(* Logix 5000 project; controller Thurs_Lab2 vendor 1 type 14 code 156 rev 30.11; software revision 30.00 *)

TASK MainTask (continuous, watchdog 500 ms) : MainProgram

MODULES
   Local : vendor 1 type 14 code 156 (Compact 0, rev 30.11)
      DC_input : 1769-IQ16 (Compact 1, rev 1.1, Input RPI 20 ms)   // Dc input
           Local:1:I.Data.0   // PB0
           Local:1:I.Data.1   // PB1
           Local:1:I.Data.2   // PB2
           Local:1:I.Data.3   // PB3
           Local:1:I.Data.4   // PB4
           Local:1:I.Data.5   // PB5
           Local:1:I.Data.6   // CYLINDER 2 NOT RETRACTED
           Local:1:I.Data.7   // MOTOR WHEEL PE
           Local:1:I.Data.8   // PART PRESENT PX
           Local:1:I.Data.9   // SPARE
           Local:1:I.Data.10   // CYLINDER 1 EXTEND PX
           Local:1:I.Data.11   // CYLINDER 1 RETRACT PX
           Local:1:I.Data.12   // CYCLE STOP
           Local:1:I.Data.13   // CYCLE START
           Local:1:I.Data.14   // ESTOP PRESSED
           Local:1:I.Data.15   // SAFETY RELAY OFF
      Relay_output : vendor 1 type 7 code 86 (Compact 3, rev 3.1, Output RPI 20 ms)   // Relay output module
           Local:3:O.Data.0   // CYLINDER 1 RETRACT
           Local:3:O.Data.1   // CYLINDER 1 EXTEND
           Local:3:O.Data.2   // CYLINDER 2 EXTEND
           Local:3:O.Data.7   // WHEEL MOTOR
           Local:3:O.Data.3   // SPARE
           Local:3:O.Data.4   // CYLINDER 3 EXTEND
           Local:3:O.Data.5   // CYLINDER 3 RETRACT
           Local:3:O.Data.6   // CYLINDER 4 EXTEND
      DC_output : 1769-OB16 (Compact 2, rev 2.1, Output RPI 20 ms)   // DC output slot
           Local:2:O.Data.0   // PL0
           Local:2:O.Data.1   // PL1
           Local:2:O.Data.2   // PL2
           Local:2:O.Data.3   // PL3
           Local:2:O.Data.4   // PL4
           Local:2:O.Data.5   // PL5
           Local:2:O.Data.6   // SPARE
           Local:2:O.Data.7   // SPARE
           Local:2:O.Data.8   // RED STACK LITE
           Local:2:O.Data.9   // YELLOW STACK LITE
           Local:2:O.Data.10   // GREEN STACK LITE
           Local:2:O.Data.11   // BLUE STACK LITE
           Local:2:O.Data.13   // SPARE
           Local:2:O.Data.14   // SPARE
           Local:2:O.Data.15   // VFD RUN
           Local:2:O.Data.12   // WHITE STACK LITE
      CELL : vendor 1 type 14 code 156 (Ethernet 192.168.0.100, rev 30.1, $565c2e57$ RPI 20 ms)
      IO : 1794-AENT (Ethernet 192.168.0.17, rev 2.12, Output RPI 20 ms)
         Real_IO : vendor 1 type 10 code 24 (Flex 0, rev 2.1, Output RPI 80 ms)
END_MODULES

TYPE CYLINDER :
STRUCT
   EXT_SIG : BOOL;
   EXT_PX : BOOL;
   RET_PX : BOOL;
   RET_SIG : BOOL;
   MAN_EXT_SIG : BOOL;
   MAN_RET_SIG : BOOL;
   EXT_TIMER : TIMER;
   RET_TIMER : TIMER;
   EXT_FAULT : BOOL;
   EXT_LIMIT : DINT;
   EXT_FAULT_COUNT : COUNTER;
END_STRUCT
END_TYPE

TYPE DRILL2 :
STRUCT
   SETTLE : TIMER;
   MOTOR : BOOL;
   UP2SPEED : TIMER;
   CYL1 : CYLINDER;
   DRILLING : TIMER;
   STOPPING : TIMER;
   CYL2 : CYLINDER;
   CLAMP : BOOL;   // EXT CYL2
   TOO_SHALLOW : BOOL;
   TOO_DEEP : BOOL;
   SHALLOW : COUNTER;
   DEEP : COUNTER;
   CYLINDERSTATUS : DINT;
END_STRUCT
END_TYPE

TYPE DRILL3 :
STRUCT
   DRILLING : TIMER;
   UP2SPEED : TIMER;
   CYL1 : CYLINDER;
   CYL2 : CYLINDER;
   SETTLE : TIMER;
   STOPPING : TIMER;
   MOTOR : BOOL;
   PV_CYL1_RET : BOOL;
   PV_CYL1_EXT : BOOL;
   PV_CYL2_EXT : BOOL;
   PV_MOTOR : BOOL;
   TOO_SHALLOW : BOOL;
   TOO_DEEP : BOOL;
   MAX_DEPTH : DINT;
   MIN_DEPTH : DINT;
   SHALLOW : COUNTER;
   DEEP : COUNTER;
   CYLINDERSTATUS : DINT;
END_STRUCT
END_TYPE

TYPE DRILL4 :
STRUCT
   SETTLE : TIMER;
   MOTOR : BOOL;
   UP2SPEED : TIMER;
   CYL1 : CYLINDER;
   DRILLING : TIMER;
   STOPPING : TIMER;
   CYL2 : CYLINDER;
   TOO_SHALLOW : BOOL;
   TOO_DEEP : BOOL;
   SHALLOW : COUNTER;
   DEEP : COUNTER;
   CYLINDERSTATUS : DINT;
END_STRUCT
END_TYPE

TYPE FROM_CELL :   // This is the FROM_CELL UDT Defining the functions as follows.
STRUCT
   STAT_A_OP : DINT;   // defines the operation that Lab Station-A Should perform
   STAT_B_OP : DINT;   // defines the operation that Lab Station-B Should perform
   STAT_C_OP : DINT;   // defines the operation that Lab Station-C Should perform
   STAT_D_OP : DINT;   // defines the operation that Lab Station-D Should perform
   STAT_E_OP : DINT;   // defines the operation that Lab Station-E Should perform
   STAT_F_OP : DINT;   // defines the operation that Lab Station-F Should perform
   STAT_G_OP : DINT;   // defines the operation that Lab Station-G Should perform
   STAT_H_OP : DINT;   // defines the operation that Lab Station-H Should perform
   STAT_I_OP : DINT;   // defines the operation that Lab Station-I Should perform
   OK2BEGIN : DINT;   // Signal that ALL Stations may begin their operation.
   OVER : DINT;   // Station 7 (consumed) bit MOVE PART to SORT IN OVER BIN
   REJECT : DINT;   // Station 7 (consumed) bit to REJECT THE PART
   UNDER : DINT;   // Station 7 (consumed) bit MOVE PART to SORT IN UNDER BIN
END_STRUCT
END_TYPE

TYPE TO_CELL :   // This is the TO_CELL UDT Defining the functions as follows.
STRUCT
   AUTO : DINT;
   BYPASS : DINT;
   DONE : DINT;
   MANUAL : DINT;
   OVER : DINT;
   REJECT : DINT;
   UNDER : DINT;
END_STRUCT
END_TYPE

VAR_GLOBAL   (* controller tags *)
   A_BLUE_STK : BOOL;
   A_CYL1_EXT : COUNTER := (PRE := 10000, CU := 1);
   A_CYL1_RET : BOOL;
   A_CYL2_EXT : BOOL;
   A_CYL2_RET : COUNTER := (PRE := 10000, CU := 1);
   A_CYL_1_EXT : BOOL;
   A_GREEN_STK : BOOL := 1;
   A_ONE_SHOT_SCAN : BOOL := 1;
   A_OUTPUT : INT;
        .4   // PL4
        .8   // RED_STK
        .12   // WHITE_STK
        .13   // SPARE
        .5   // PL5
        .10   // GREEN_STK
        .11   // BLUE_STK
        .6   // SPARE
        .9   // YELLOW_STK
        .0   // PL0
        .1   // PL1
        .2   // PL2
        .3   // PL3
        .14   // SPARE
        .15   // VFD RUN
        .7   // SPARE
   A_PL0 : BOOL;
   A_PL1 : BOOL;
   A_PL2 : BOOL;
   A_PL3 : BOOL;
   A_PL4 : BOOL;
   A_PL5 : BOOL;
   A_RED_STK : BOOL;
   A_REJECT_MAX : DINT;
   A_REJECT_MIN : DINT;
   A_REL_OUT : SINT;
        .0   // CYL_1_RET
        .1   // CYL_1_EXT
        .2   // CYL_2_EXT
        .3   // SPARE
        .4   // CYL_3_EXT
        .5   // CYL_3_RET
        .6   // CYL_4_EXT
        .7   // WHEEL MOTOR
   A_Timer_Ret : TIMER := (PRE := 500000);
   A_VFD_RUN : BOOL;
   A_WHEEL_MOTOR : BOOL;
   A_WHITE_STK : BOOL;
   A_YELLOW_STK : BOOL := 1;
   ALARM_CLOSE : BOOL := 1;
   ANTI_REPEAT : BOOL;
   ANTI_REPEAT_ONE_SHOT_SCAN : BOOL;
   AUTO : BOOL := 1;
   AUTO_DISABLE : BOOL;
   Auto_ONE_SHOT_SCAN : BOOL;
   AVERAGE : DINT;
   AVG : DINT;
   BLINK : TIMER := (PRE := 500);
   BLINK_PL1 : TIMER := (PRE := 1000);
   BLINK_PL3 : TIMER := (PRE := 1000);
   BLINK_TIMER : TIMER := (PRE := 1000);
   BLINKOFF : TIMER := (PRE := 500, ACC := 480, EN := 1, TT := 1);
   BLINKON : TIMER := (PRE := 500);
   BLUE : BOOL;
   BLUE_4_OVERSIZED : BOOL;
   BLUE_BLINKER : TIMER := (PRE := 1000);
   BLUE_STACK_LITE : BOOL := 1;
   BLUE_STK : BOOL := 1;
   BUTTON : BOOL;
   BYPASS : BOOL;
   CHECK_0 : BOOL;
   CHECK_1 : BOOL;
   CONTINUE : BOOL;
   CONTROL : CONTROL := (LEN := 10);
   CONV1_WHEEL_MOTOR : BOOL;
   COUNTER : COUNTER := (PRE := 10000);
   CYCLE_COUNT : COUNTER := (PRE := 5, ACC := 1);
   CYCLE_START : BOOL;
   CYCLE_STOP : BOOL := 1;
   CYCLE_TIME : TIMER := (PRE := 10000000, ACC := 58718, EN := 1, TT := 1);
   CYL1_EXT : COUNTER := (PRE := 10000, CU := 1);
   CYL1_EXT_4_SORTING : BOOL;
   CYL1_EXT_4_TEST : BOOL;
   CYL1_EXT_COUNT : COUNTER := (PRE := 10, CU := 1);
   CYL1_EXT_COUNTMOVER : BOOL := 1;
   CYL1_EXT_IN_SORT_OP : BOOL;
   CYL1_EXT_IN_TEST_OP : BOOL;
   CYL1_EXT_PX : BOOL;
   CYL1_EXT_PX_VALUE : DINT;
   CYL1_EXT_SUM : DINT;
   CYL1_EXTEND : BOOL;
   CYL1_RET : BOOL;
   CYL1_RET_4_SORTING : BOOL;
   CYL1_RET_4_TEST : BOOL;
   CYL1_RET_IN_SORT_OP : BOOL;
   CYL1_RET_IN_TEST_OP : BOOL;
   CYL1_RET_PX : BOOL := 1;
   CYL2_EXT : BOOL;
   CYL2_EXT_4_LOAD_AND_UNLOAD : BOOL := 1;
   CYL2_EXT_4_LOADING : BOOL;
   CYL2_EXT_4_SORTING : BOOL;
   CYL2_EXT_PX : BOOL;
   CYL2_NOT_RET : BOOL;
   CYL2_NOT_RET_PX : BOOL;
   CYL2_RET : COUNTER := (PRE := 10000, ACC := 1, CU := 1);
   CYL2_RET_4_UNLOADING : BOOL;
   CYL2_RET_PX : BOOL;
   CYL3_EXT : BOOL;
   CYL3_RET : BOOL;
   CYL4_EXT : BOOL;
   CYLINDER1 : CYLINDER;
   CYLINDER1_EXTEND : BOOL;
   CYLINDER1_EXTEND_PX : BOOL;
   CYLINDER1_RETRACT : BOOL;
   CYLINDER1_RETRACT_PX : BOOL;
   CYLINDER2_EXTEND : BOOL := 1;
   CYLINDERSTATUS : DINT := 2;
   DEEP : COUNTER := (PRE := 1000, CU := 1);
   DELAY_1 : TIMER := (PRE := 1000);
   DELAY_PE_INPUT : TIMER := (PRE := 500);
   DELAY_PE_INPUT_PSB : TIMER := (PRE := 500);
   DELAY_PE_INPUT_PSW : TIMER := (PRE := 500);
   DELAY_PE_INPUT_STATE : TIMER := (PRE := 500);
   DONE_MOV : BOOL;
   DRILL2 : DRILL2 := (SETTLE.PRE := 500, UP2SPEED.PRE := 1000, CYL1.RET_PX := 1, CYL1.EXT_TIMER.PRE := 10000, CYL1.EXT_LIMIT := 1500, DRILLING.PRE := 2000, STOPPING.PRE := 2000, SHALLOW.PRE := 1000, DEEP.PRE := 1000);
   DRILL3 : DRILL3 := (DRILLING.PRE := 2000, UP2SPEED.PRE := 1000, CYL1.RET_PX := 1, CYL1.EXT_TIMER.PRE := 10000, CYL1.EXT_LIMIT := 1500, STOPPING.PRE := 2000, MAX_DEPTH := 22000, MIN_DEPTH := 20000, SHALLOW.PRE := 1000, DEEP.PRE := 1000);
   DRILL4 : DRILL4 := (SETTLE.PRE := 500, UP2SPEED.PRE := 1000, CYL1.RET_PX := 1, CYL1.EXT_TIMER.PRE := 10000, CYL1.EXT_LIMIT := 1500, DRILLING.PRE := 2000, STOPPING.PRE := 2000, SHALLOW.PRE := 1000, SHALLOW.ACC := 10, SHALLOW.CU := 1, DEEP.PRE := 1000);
   ESTOP : BOOL;
   ESTOP_PRESSED : BOOL;
   Ext_Fault_Lim : DINT := 1500;
   EXTEND : TIMER := (PRE := 5000);
   EXTEND_CYL1 : BOOL;
   EXTEND_CYL2 : BOOL;
   ExtendFault : BOOL;
   FAILURE2LOAD : TIMER := (PRE := 8000);
   FAILURE_2_LOAD : BOOL;
   FAULT : BOOL;
   FAULT_4_FAILURE2LOAD : BOOL;
   FAULT_4_PART_REJECT : BOOL;
   FAULT_4_UNDERSIZE_PART : BOOL;
   FAULT_4_UNDERSIZED_PART : BOOL;
   FAULT_COUNTER : COUNTER := (PRE := 1000000);
   FAULT_FAILURE2LOAD : BOOL;
   FAULT_PART_REJECT : BOOL;
   FAULT_RESET_COUNT : COUNTER := (PRE := 100000, ACC := 37);
   FAULT_S : DINT;
   FAULTED : BOOL;
   FLASHER_GREEN : TIMER := (PRE := 500, ACC := 334);
   FROM_CELL : FROM_CELL := (STAT_A_OP := 1, STAT_B_OP := 1, STAT_C_OP := 8, STAT_D_OP := 1, STAT_E_OP := 7, STAT_F_OP := 8, STAT_G_OP := 7, STAT_H_OP := 4, STAT_I_OP := 2);
   GGG : DINT;
   GOOD_PART : BOOL;
   GOODPART : DINT;
   GOODSIZE_MAX : DINT := 20000;
   GOODSIZE_MIN : DINT := 10000;
   GREEN_4_GOOD : BOOL;
   GREEN_BLINKER : TIMER := (PRE := 1000);
   GREEN_STACK_LITE : BOOL := 1;
   GREEN_STK : BOOL := 1;
   HOLE_DEPTH : DINT;
   HOLE_DEPTH_MAX : DINT := 27500;
   HOLE_DEPTH_MIN : DINT := 22500;
   HOLE_SHALLOW_MAX : DINT := 8000;
   HOLE_SHALLOW_MIN : DINT := 160;
   INPUT : INT := -9921;
        .0   // PB0
        .2   // PB2
        .6   // CYL_2_NOT_ RET
        .7   // MOTOR WHEEL PE
        .1   // PB1
        .3   // PB3
        .4   // PB4
        .5   // PB5
        .8   // PART PRESENT PX
        .9   // SPARE
        .10   // CYL_1_EXT_PX
        .11   // CYL_1_RET_PX
        .12   // CYCLE STOP
        .13   // CYCLE START
        .14   // ESTOP PRESSED
        .15   // SAFETY RELAY OFF
   LASERPE : DINT := 23792;
   LAST_CYCLE_COUNT : COUNTER := (PRE := 1);
   LAST_CYCLE_TIME : DINT;
   LIMIT_PSB : BOOL;
   LIMIT_PSW : BOOL;
   LIMIT_STATE : BOOL;
   LOAD_ONE_SHOT_SCAN : BOOL;
   LOAD_ONE_SHOT_SCAN_1 : BOOL;
   LOAD_ONE_SHOT_SCAN_2 : BOOL;
   LOAD_ONE_SHOT_SCAN_3 : BOOL;
   LOAD_STEP : DINT;
   LOAD_WHITE_STK : BOOL;
   LOADING : BOOL;
   M_BLUE_STK : BOOL;
   M_CYL1_EXT : COUNTER := (PRE := 10000);
   M_CYL1_RET : BOOL;
   M_CYL2_EXT : BOOL;
   M_CYL2_RET : COUNTER := (PRE := 10000, ACC := 1);
   M_CYL_1_EXT : BOOL;
   M_GREEN_STK : BOOL;
   M_ONE_SHOT_SCAN : BOOL;
   M_OUTPUT : INT;
        .0   // PL0
        .13   // SPARE
        .14   // SPARE
        .1   // PL1
        .2   // PL2
        .3   // PL3
        .4   // PL4
        .6   // SPARE
        .12   // WHITE_STK
        .15   // VFD RUN
        .10   // GREEN_STK
        .8   // RED_STK
        .5   // PL5
        .9   // YELLOW_STK
        .11   // BLUE_STK
        .7   // SPARE
   M_PL0 : BOOL;
   M_PL1 : BOOL;
   M_PL2 : BOOL;
   M_PL3 : BOOL;
   M_PL4 : BOOL;
   M_PL5 : BOOL;
   M_PLO : BOOL;
   M_RED_STK : BOOL;
   M_REL_OUT : SINT;
        .0   // CYL_1_RET
        .1   // CYL_1_EXT
        .2   // CYL_2_EXT
        .3   // SPARE
        .4   // CYL_3_EXT
        .5   // CYL_3_RET
        .6   // CYL_4_EXT
        .7   // WHEEL MOTOR
   M_System_Enable : BOOL;
   M_Timer_Ret : TIMER := (PRE := 500000);
   M_WHEEL_MOTOR : BOOL;
   M_WHITE_STK : BOOL;
   M_YELLOW_STK : BOOL;
   MACHINE_PAUSED : BOOL;
   Man_ONE_SHOT_SCAN : BOOL := 1;
   Manual : BOOL;
   MARK_BLUE : BOOL;
   MARK_CYL1 : CYLINDER := (RET_PX := 1);
   MARK_CYL1_EXT_PX : BOOL;
   MARK_GREEN : BOOL;
   MARK_LIGHTS : BOOL;
   MARK_ONE_SHOT_SCAN : BOOL;
   MARK_RED : BOOL;
   MARK_WHITE_STK : BOOL;
   MARK_YELLOW : BOOL;
   MASTER_RESET_COUNT : COUNTER := (PRE := 2);
   MASTER_RESET_COUNT1 : COUNTER := (PRE := 2);
   MASTER_RESET_COUNT2 : COUNTER := (PRE := 2);
   MASTER_RESET_COUNT3 : COUNTER := (PRE := 2);
   MASTER_RESET_COUNT4 : COUNTER := (PRE := 2);
   MASTER_RESET_COUNT5 : COUNTER := (PRE := 2);
   MASTER_RESET_COUNT6 : COUNTER := (PRE := 2);
   MASTER_RESET_COUNT7 : COUNTER := (PRE := 2);
   MODE_SELECT : DINT := 1;
   MOTOR_QUARTER_REVS : COUNTER;
   MOTOR_WHEEL : BOOL;
   MOTOR_WHEEL_PE : BOOL := 1;
   MSTER_RESET_TWCE : BOOL;
   NOT_values : DINT;
   ONE_SHOT2 : BOOL;
   ONE_SHOT_0 : BOOL;
   ONE_SHOT_1 : BOOL;
   ONE_SHOT_10 : BOOL;
   ONE_SHOT_2 : BOOL;
   ONE_SHOT_3 : BOOL;
   ONE_SHOT_4 : BOOL;
   ONE_SHOT_6 : BOOL;
   ONE_SHOT_7 : BOOL;
   ONE_SHOT_8 : BOOL;
   ONE_SHOT_ENABLE : BOOL;
   ONE_SHOT_PSB0 : BOOL;
   ONE_SHOT_PSB1 : BOOL;
   ONE_SHOT_PSW0 : BOOL := 1;
   ONE_SHOT_PSW1 : BOOL := 1;
   ONE_SHOT_SCAN : BOOL;
   ONE_SHOT_STATE0 : BOOL;
   ONE_SHOT_STATE1 : BOOL;
   ONE_SHOT_TEST : BOOL;
   ONESHOT1 : BOOL;
   ONESHOT2 : BOOL;
   ONESHOT3 : BOOL;
   ONESHOT4 : BOOL := 1;
   ONESHOT_0 : BOOL := 1;
   ONESHOT_0_PSW : BOOL;
   ONESHOT_1 : BOOL := 1;
   ONESHOT_1_PSW : BOOL;
   OP1_CYL2_EXT : BOOL;
   OP1_STOP : BOOL;
   OP2_ONE_SHOT_SCAN : BOOL;
   OP2_STEP : DINT;
   OP2_STOP : BOOL;
   OP2STEP : DINT := 3;
   OP3_ONE_SHOT_SCAN : BOOL;
   OP3_STOP : BOOL;
   OP4_ONE_SHOT_SCAN : BOOL;
   OP4_STOP : BOOL;
   OP5_REJECT : DINT := 1;
   OP5_STATIC_GOOD : BOOL;
   OP5_STATIC_OVER : BOOL;
   OP5_STATIC_REJECT : BOOL;
   OP5_STATIC_UNDER : BOOL;
   OP5_STOP : BOOL;
   OP5_TEST : DINT := 2;
   OP5_TEST_STATIC : DINT := 3;
   OP6_MARK : TIMER := (PRE := 4000);
   OP6_OP7 : DINT := 3;
   OP6_STOP : BOOL;
   OP6MARK : FBD_TIMER;
   OP7_SORT : DINT := 3;
   OP7_STOP : BOOL;
   OP8_BLUE_STK : BOOL;
   OP8_GRN_STK : BOOL;
   OP8_RED_STK : BOOL;
   OP8_YELLOW_STK : BOOL;
   OPERATION : DINT := 2;
   OPERATION_5_OVER : BOOL;
   OPERATION_5_REJECT : BOOL;
   OPERATION_5_UNDER : BOOL;
   OPERATION_7_OVER : BOOL;
   OPERATION_7_REJECT : BOOL;
   OPERATION_7_UNDER : BOOL;
   OPERATION_DONE : DINT;
   OPERATION_OFF : DINT := 2;
   Oring : DINT := 1007;
   OUT_OF_INK_FAULT : BOOL;
   OUTPUT : INT;
        .0   // PL0
        .1   // PL1
        .10   // GREEN_STK
        .11   // BLUE_STK
        .12   // WHITE_STK
        .13   // SPARE
        .14   // SPARE
        .15   // VFD RUN
        .2   // PL2
        .3   // PL3
        .4   // PL4
        .5   // PL5
        .6   // SPARE
        .7   // SPARE
        .8   // RED_STK
        .9   // YELLOW_STK
   OVERSIZE_HIGH : DINT := 30000;
   OVERSIZE_LOW : DINT := 19990;
   OVERSIZE_STEP : DINT;
   OVERSIZE_STEP_0 : BOOL;
   PART_NOT_PX : BOOL;
   PART_PRESENT_PX : BOOL := 1;
   PART_PX : BOOL := 1;
   PARTS : COUNTER := (PRE := 1000);
   PARTS_COUNT_TOTALIZER : COUNTER := (PRE := 100000);
   PAUSE : BOOL;
   PAUSED : BOOL;
   PAUSED_OPERATION_1 : BOOL;
   PAUSED_OPERATION_5 : BOOL;
   PAUSED_OPERATION_7 : BOOL;
   PB0 : BOOL;
   PB1 : BOOL;
   PB1_ON : DINT;
   PB2 : BOOL;
   PB3 : BOOL;
   PB4 : BOOL;
   PB5 : BOOL;
   PB_RESET_FAULT : BOOL;
   PILOT_LIGHT_0 : BOOL;
   PILOT_LIGHT_1 : BOOL;
   PILOT_LIGHT_2 : BOOL;
   PILOT_LIGHT_3 : BOOL;
   PILOT_LIGHT_4 : BOOL;
   PILOT_LIGHT_5 : BOOL;
   PL1 : BOOL;
   PL1_BLINKER : TIMER := (PRE := 1000);
   PL3 : BOOL;
   PL_CONTROL : DINT := 55;
   PPPPPPP : DINT;
   PREVENT_FAULT_5 : DINT;
   PREVENT_FAULT_7 : DINT;
   PRODUCTION_ONE_SHOT : BOOL;
   PUSH : BOOL;
   PUSH_BUTTON_0 : BOOL;
   PV_ANALOG_PROBE : DINT := 12400;
   PV_ANALOG_PROBE_STATIC : DINT := 4150;
   PV_AUTO : BOOL := 1;
   PV_CONV1_WHEEL_MOTOR : BOOL;
   PV_CYL1_DEPTH : DINT := 144;
   PV_CYL1_EXT : BOOL;
   PV_CYL1_EXT_LIMIT : DINT := 1500;
   PV_CYL1_EXT_SIG : BOOL;
   PV_CYL1_EXT_TIME : DINT := 615;
   PV_CYL1_RET : BOOL;
   PV_CYL1_RET_SIG : BOOL;
   PV_CYL2_EXT : BOOL;
   PV_CYL2_EXT_SIG : BOOL;
   PV_DISPLAY_MODE : DINT;
   PV_DRILLING : DINT := 2000;
   PV_FAULT_COUNT_RESET : BOOL;
   PV_FAULT_RESET : BOOL;
   PV_HOLE_TOO_DEEP : DINT := 25000;
   PV_HOLE_TOO_SHALLOW : DINT := 800;
   PV_LAST_CYCLE_TIME : DINT;
   PV_LAST_CYCLE_TIME1 : DINT;
   PV_LAST_CYCLE_TIME2 : DINT;
   PV_LAST_CYCLE_TIME3 : DINT;
   PV_LAST_CYCLE_TIME4 : DINT;
   PV_LAST_CYCLE_TIME5 : DINT;
   PV_MAX_DEPTH : DINT := 4300;
   PV_MIN_DEPTH : DINT := 300;
   PV_MOTOR_START : BOOL;
   PV_OP1 : BOOL;
   PV_OP5 : BOOL;
   PV_OP5_PROBE_VALUE : DINT;
   PV_OP7 : BOOL;
   PV_OP_SELECT : DINT;
   PV_PARTS_COUNT_RESET : BOOL;
   PV_RESET : BOOL;
   PV_RESET_FAULT : BOOL;
   PV_STOPPING : DINT := 2000;
   PV_UP2SPEED : DINT := 1000;
   READY_TO_INDEX : BOOL;
   RED_4_UNDERSIZED : BOOL;
   RED_BLINKER : TIMER := (PRE := 1000);
   RED_STACK_LITE : BOOL;
   RED_STK : BOOL;
   REJECT_FAULT : BOOL;
   REJECT_STEP : DINT;
   REJECT_STEP_0 : BOOL;
   REL_OUT : SINT;
        .1   // CYL_1_EXT
        .2   // CYL_2_EXT
        .4   // CYL_3_EXT
        .0   // CYL_1_RET
        .7   // WHEEL MOTOR
        .3   // SPARE
        .5   // CYL_3_RET
        .6   // CYL_4_EXT
   RELEASE : DINT;
   RESET : BOOL;
   RESET_CELL_TAGS : BOOL;
   RESET_FAULT : BOOL;
   RESET_OVER_5 : BOOL;
   RESET_PB : BOOL;
   RESET_REJECT_5 : BOOL;
   RESET_UNDER_5 : BOOL;
   RETRACT_CYL1 : BOOL;
   REVOLUTIONS : COUNTER := (PRE := 12);
   RUN_DC_MOTOR : BOOL;
   SAFETY_RELAY_OFF : BOOL;
   SEQ_A_TO_D_COMPLETE : BOOL;
   SEQ_EN : BOOL := 1;
   SETSPEED7 : DINT := 5000;
   SETTLE1 : TIMER := (PRE := 5000);
   SETTLE5 : TIMER := (PRE := 2000);
   SHALLOW : COUNTER := (PRE := 1000, ACC := 1, CU := 1);
   SORT_ONE_SHOT_SCAN : BOOL;
   SORT_SEQ_FOR_REJECT : DINT;
   SORT_STEP : DINT;
   SPARE : BOOL;
   STA : DINT;
   START_SEQ : BOOL;
   START_SIGNAL : BOOL;
   START_SORT_SEQUENCE : BOOL;
   START_TEST_SEQ : BOOL;
   START_UNLOAD_LOAD_SEQ : BOOL;
   STATB_OP : DINT;
   STATE : DINT;
   STATUS : DINT := 3;
   STEP : DINT := 1;
   Step1 : DINT := -239;
   Step2 : DINT := 301989887;
   Step3 : DINT := 255;
   STEP_01 : SEQ_STEP;
   StoreExt : DINT[10];
   SYS_ENABLE : BOOL;
   System_Enable : BOOL := 1;
   T : DINT;
   T0 : BOOL;
   T1 : BOOL;
   T2 : BOOL;
   T_Motor : TIMER := (PRE := 500000);
   TEST_ONE_SHOT_SCAN : BOOL;
   TEST_STEP : DINT;
   Timer : TIMER := (PRE := 500000);
   TIMER_1 : TIMER := (PRE := 500);
   TIMER_2 : TIMER := (PRE := 500);
   TIMER_CELL_DONE : TIMER := (PRE := 1000);
   Timer_Non_Ret : TIMER := (PRE := 3000);
   Timer_Ret : TIMER := (PRE := 500000);
   TO_CELL : TO_CELL := (AUTO := 1); {produced}
   TO_CELL_GOOD_PART : BOOL;
   TO_CELL_GOODPART : BOOL;
   TO_CELL_OVER : BOOL;
   TO_CELL_REJECT : BOOL;
   TO_CELL_UNDER : BOOL;
   TOO_DEEP : BOOL;
   TOO_SHALLOW : BOOL;
   TRANSFER7 : TIMER := (PRE := 10000);
   TRANSFER7_TIME_EXCEED : BOOL;
   TWO_HAND_START : BOOL;
   UNDERSIZE_HIGH : DINT := 9990;
   UNDERSIZE_LOW : DINT := 3000;
   UNDERSIZE_STEP : DINT;
   UNDERSIZE_STEP_0 : BOOL;
   UNLOAD_SCAN : BOOL;
   UNLOADING : BOOL;
   UP2SPEED7 : TIMER := (PRE := 1000);
   WHEEL_MOTOR : BOOL;
   WHEEL_PE : COUNTER := (PRE := 64, CU := 1);
   WHITE_STACK_LITE : BOOL := 1;
   WHITE_STK : BOOL := 1;
   Xoring : DINT := 238;
   YELLOW_4_REJECTION : BOOL;
   YELLOW_STACK_LITE : BOOL;
   YELLOW_STK : BOOL;
   ZEROSPEED7 : TIMER := (PRE := 5000);
END_VAR

PROGRAM MainProgram   (* main routine MainRoutine *)
VAR
   Action_000 : SFC_ACTION := (Status := 16#0020_0000, PauseTimer := 1);
   Action_001 : SFC_ACTION := (Status := 16#0020_0000, PauseTimer := 1);
   Action_002 : SFC_ACTION := (Status := 16#0020_0000, PauseTimer := 1);
   Action_003 : SFC_ACTION := (Status := 16#0020_0000, PauseTimer := 1);
   Action_004 : SFC_ACTION := (Status := 16#0020_0000, PauseTimer := 1);
   Action_005 : SFC_ACTION := (Status := 16#0020_0000, PauseTimer := 1);
   Action_006 : SFC_ACTION := (Status := 16#0020_0000, PauseTimer := 1);
   Action_007 : SFC_ACTION := (Status := 16#0020_0000, PauseTimer := 1);
   Action_008 : SFC_ACTION := (Status := 16#0020_0000, PauseTimer := 1);
   Action_009 : SFC_ACTION := (Status := 16#0020_0000, PauseTimer := 1);
   Action_010 : SFC_ACTION := (Status := 16#0020_0000, PauseTimer := 1);
   Action_011 : SFC_ACTION := (Status := 16#0020_0000, PauseTimer := 1);
   Action_012 : SFC_ACTION := (Status := 16#0020_0000, PauseTimer := 1);
   Action_013 : SFC_ACTION := (Status := 16#0020_0000, PauseTimer := 1);
   Action_014 : SFC_ACTION := (Status := 16#0020_0000, PauseTimer := 1);
   Action_015 : SFC_ACTION := (Status := 16#c020_0000, A := 1, Q := 1, PauseTimer := 1, Count := 1);
   Action_016 : SFC_ACTION := (Status := 16#c020_0000, A := 1, Q := 1, PauseTimer := 1, Count := 1);
   Action_017 : SFC_ACTION := (Status := 16#c020_0000, A := 1, Q := 1, PauseTimer := 1, Count := 1);
   Action_018 : SFC_ACTION := (Status := 16#c020_0000, A := 1, Q := 1, PauseTimer := 1, Count := 1);
   Action_019 : SFC_ACTION := (Status := 16#c020_0000, A := 1, Q := 1, PauseTimer := 1, Count := 1);
   Action_020 : SFC_ACTION := (Status := 16#c020_0000, A := 1, Q := 1, PauseTimer := 1, Count := 1);
   Action_021 : SFC_ACTION := (Status := 16#c020_0000, A := 1, Q := 1, PauseTimer := 1, Count := 1);
   Action_022 : SFC_ACTION := (Status := 16#c020_0000, A := 1, Q := 1, PauseTimer := 1, Count := 1);
   Action_023 : SFC_ACTION := (Status := 16#c020_0000, A := 1, Q := 1, PauseTimer := 1, Count := 1);
   Action_024 : SFC_ACTION := (Status := 16#c020_0000, A := 1, Q := 1, PauseTimer := 1, Count := 1);
   BAND_01 : FBD_BOOLEAN_AND := (In2 := 1, In4 := 1, In5 := 1, In6 := 1, In7 := 1, In8 := 1);
   BAND_02 : FBD_BOOLEAN_AND := (In2 := 1, In3 := 1, In4 := 1, In5 := 1, In6 := 1, In7 := 1, In8 := 1);
   BNOT_01 : FBD_BOOLEAN_NOT := (Out := 1);
   BNOT_02 : FBD_BOOLEAN_NOT := (In := 1);
   BNOT_03 : FBD_BOOLEAN_NOT := (Out := 1);
   BNOT_04 : FBD_BOOLEAN_NOT := (Out := 1);
   STEP0 : SFC_STEP := (Status := 16#0020_0000, PauseTimer := 1);
   STEP1 : SFC_STEP := (Status := 16#0020_0000, PauseTimer := 1);
   STEP2 : SFC_STEP := (Status := 16#0020_0000, PauseTimer := 1);
   STEP3 : SFC_STEP := (Status := 16#0020_0000, PauseTimer := 1);
   STEP4 : SFC_STEP := (Status := 16#0020_0000, PauseTimer := 1);
   Step_000 : SFC_STEP := (Status := 16#0820_0201, DN := 1, PauseTimer := 1, T := 436961, TMax := 436961, Count := 1);
   Step_001 : SFC_STEP := (Status := 16#0020_0000, PauseTimer := 1);
   Step_002 : SFC_STEP := (Status := 16#0020_0000, PauseTimer := 1);
   Step_003 : SFC_STEP := (Status := 16#0020_0000, PauseTimer := 1);
   Step_004 : SFC_STEP := (Status := 16#0020_0000, PauseTimer := 1);
   Step_005 : SFC_STEP := (Status := 16#0020_0000, PauseTimer := 1);
   Step_006 : SFC_STEP := (Status := 16#0020_0000, PauseTimer := 1);
   Step_007 : SFC_STEP := (Status := 16#0020_0000, PauseTimer := 1);
   Step_008 : SFC_STEP := (Status := 16#0020_0000, PauseTimer := 1);
   Step_009 : SFC_STEP := (Status := 16#0020_0000, PauseTimer := 1);
   Step_010 : SFC_STEP := (Status := 16#0020_0000, PauseTimer := 1);
   Step_011 : SFC_STEP := (Status := 16#a820_0001, X := 1, SA := 1, DN := 1, PauseTimer := 1, T := 68777, TMax := 68777, Count := 1);
   Step_012 : SFC_STEP := (Status := 16#a820_0001, X := 1, SA := 1, DN := 1, PauseTimer := 1, T := 68777, TMax := 68777, Count := 1);
   Step_013 : SFC_STEP := (Status := 16#a820_0001, X := 1, SA := 1, DN := 1, PauseTimer := 1, T := 68777, TMax := 68777, Count := 1);
   Step_014 : SFC_STEP := (Status := 16#0020_0000, PauseTimer := 1);
   Step_015 : SFC_STEP := (Status := 16#a820_0001, X := 1, SA := 1, DN := 1, PauseTimer := 1, T := 68777, TMax := 68777, Count := 1);
   Step_016 : SFC_STEP := (Status := 16#a820_0001, X := 1, SA := 1, DN := 1, PauseTimer := 1, T := 68777, TMax := 68777, Count := 1);
   Step_017 : SFC_STEP := (Status := 16#a820_0001, X := 1, SA := 1, DN := 1, PauseTimer := 1, T := 68777, TMax := 68777, Count := 1);
   Step_018 : SFC_STEP := (Status := 16#a820_0001, X := 1, SA := 1, DN := 1, PauseTimer := 1, T := 68777, TMax := 68777, Count := 1);
   Step_019 : SFC_STEP := (Status := 16#a820_0001, X := 1, SA := 1, DN := 1, PauseTimer := 1, T := 68777, TMax := 68777, Count := 1);
   Step_020 : SFC_STEP := (Status := 16#a820_0001, X := 1, SA := 1, DN := 1, PauseTimer := 1, T := 68777, TMax := 68777, Count := 1);
   Step_021 : SFC_STEP := (Status := 16#a820_0001, X := 1, SA := 1, DN := 1, PauseTimer := 1, T := 68776, TMax := 68776, Count := 1);
   Tran_000 : BOOL := 1;
   Tran_001 : BOOL;
   Tran_002 : BOOL;
   Tran_003 : BOOL;
   Tran_004 : BOOL;
   Tran_005 : BOOL;
   Tran_006 : BOOL;
   Tran_007 : BOOL;
   Tran_008 : BOOL;
   Tran_009 : BOOL;
   Tran_010 : BOOL;
   Tran_011 : BOOL;
   Tran_012 : BOOL;
   Tran_013 : BOOL;
   Tran_014 : BOOL;
   Tran_015 : BOOL;
   Tran_016 : BOOL;
   Tran_017 : BOOL;
   Tran_018 : BOOL;
   Tran_019 : BOOL;
   Tran_020 : BOOL;
   Tran_021 : BOOL;
   Tran_022 : BOOL;
   Tran_023 : BOOL;
   Tran_024 : BOOL;
   Tran_025 : BOOL;
   Tran_027 : BOOL;
END_VAR

ROUTINE CELL   (* ladder *)
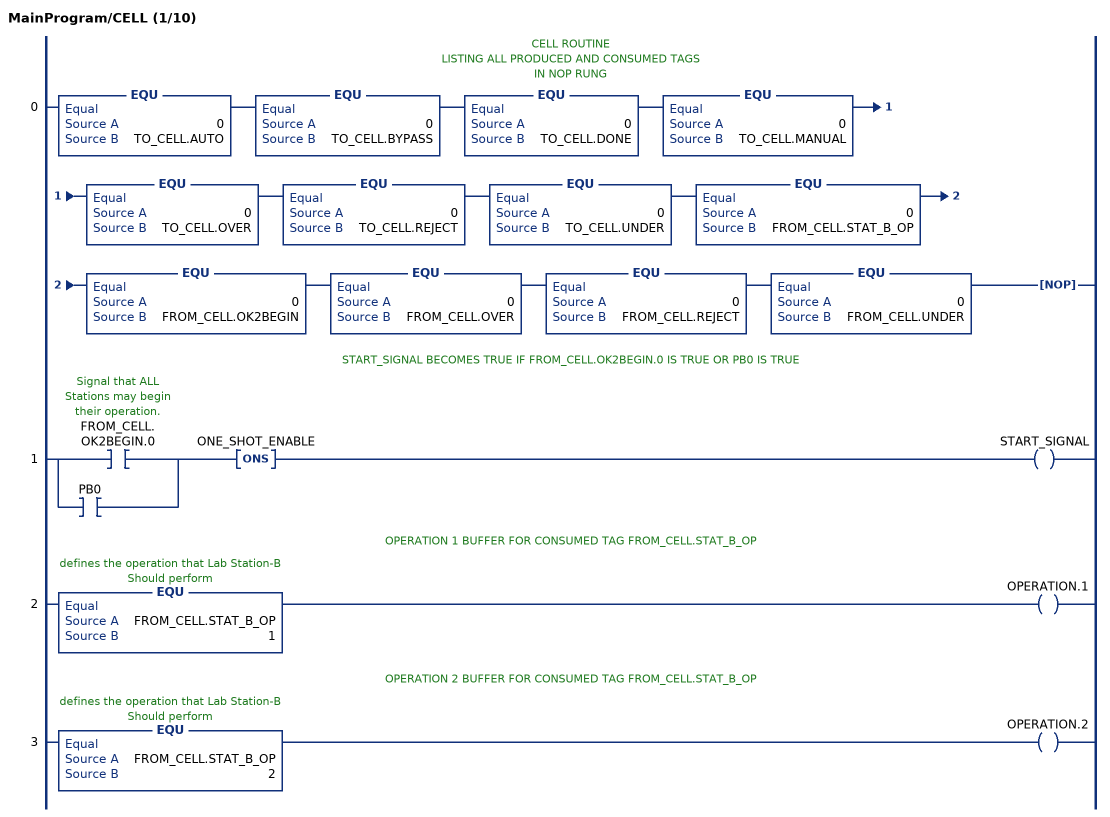
   // CELL ROUTINE
   // LISTING ALL PRODUCED AND CONSUMED TAGS
   //  IN NOP RUNG
   0: EQU(0,TO_CELL.AUTO)EQU(0,TO_CELL.BYPASS)EQU(0,TO_CELL.DONE)EQU(0,TO_CELL.MANUAL)EQU(0,TO_CELL.OVER)EQU(0,TO_CELL.REJECT)EQU(0,TO_CELL.UNDER)EQU(0,FROM_CELL.STAT_B_OP)EQU(0,FROM_CELL.OK2BEGIN)EQU(0,FROM_CELL.OVER)EQU(0,FROM_CELL.REJECT)EQU(0,FROM_CELL.UNDER)NOP();
   // START_SIGNAL BECOMES TRUE IF FROM_CELL.OK2BEGIN.0 IS TRUE OR PB0 IS TRUE
   1: [XIC(FROM_CELL.OK2BEGIN.0) ,XIC(PB0) ]ONS(ONE_SHOT_ENABLE)OTE(START_SIGNAL);
   // OPERATION 1 BUFFER FOR CONSUMED TAG FROM_CELL.STAT_B_OP
   2: EQU(FROM_CELL.STAT_B_OP,1)OTE(OPERATION.1);
   // OPERATION 2 BUFFER FOR CONSUMED TAG FROM_CELL.STAT_B_OP
   3: EQU(FROM_CELL.STAT_B_OP,2)OTE(OPERATION.2);
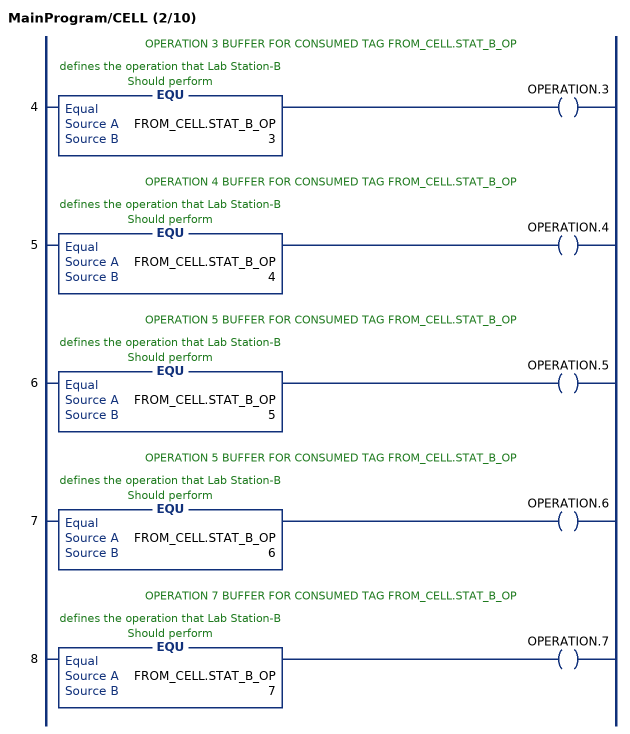
   // OPERATION 3 BUFFER FOR CONSUMED TAG FROM_CELL.STAT_B_OP
   4: EQU(FROM_CELL.STAT_B_OP,3)OTE(OPERATION.3);
   // OPERATION 4 BUFFER FOR CONSUMED TAG FROM_CELL.STAT_B_OP
   5: EQU(FROM_CELL.STAT_B_OP,4)OTE(OPERATION.4);
   // OPERATION 5 BUFFER FOR CONSUMED TAG FROM_CELL.STAT_B_OP
   6: EQU(FROM_CELL.STAT_B_OP,5)OTE(OPERATION.5);
   // OPERATION 5 BUFFER FOR CONSUMED TAG FROM_CELL.STAT_B_OP
   7: EQU(FROM_CELL.STAT_B_OP,6)OTE(OPERATION.6);
   // OPERATION 7 BUFFER FOR CONSUMED TAG FROM_CELL.STAT_B_OP
   8: EQU(FROM_CELL.STAT_B_OP,7)OTE(OPERATION.7);
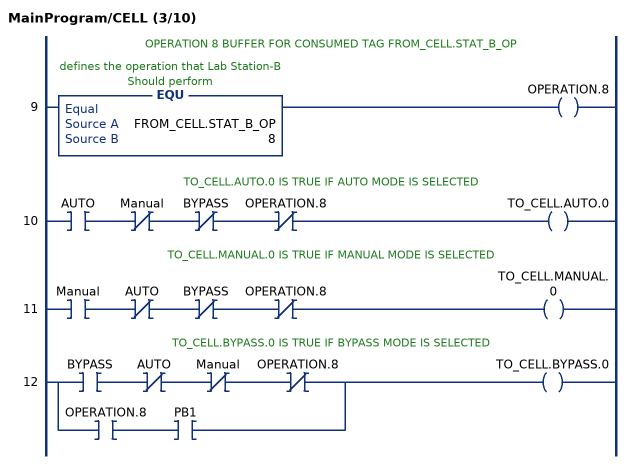
   // OPERATION 8 BUFFER FOR CONSUMED TAG FROM_CELL.STAT_B_OP
   9: EQU(FROM_CELL.STAT_B_OP,8)OTE(OPERATION.8);
   // TO_CELL.AUTO.0 IS TRUE IF AUTO MODE IS SELECTED
   10: XIC(AUTO)XIO(Manual)XIO(BYPASS)XIO(OPERATION.8)OTE(TO_CELL.AUTO.0);
   // TO_CELL.MANUAL.0 IS TRUE IF MANUAL MODE IS SELECTED
   11: XIC(Manual)XIO(AUTO)XIO(BYPASS)XIO(OPERATION.8)OTE(TO_CELL.MANUAL.0);
   // TO_CELL.BYPASS.0 IS TRUE IF BYPASS MODE IS SELECTED
   12: [XIC(BYPASS) XIO(AUTO) XIO(Manual) XIO(OPERATION.8) ,XIC(OPERATION.8) XIC(PB1) ]OTE(TO_CELL.BYPASS.0);
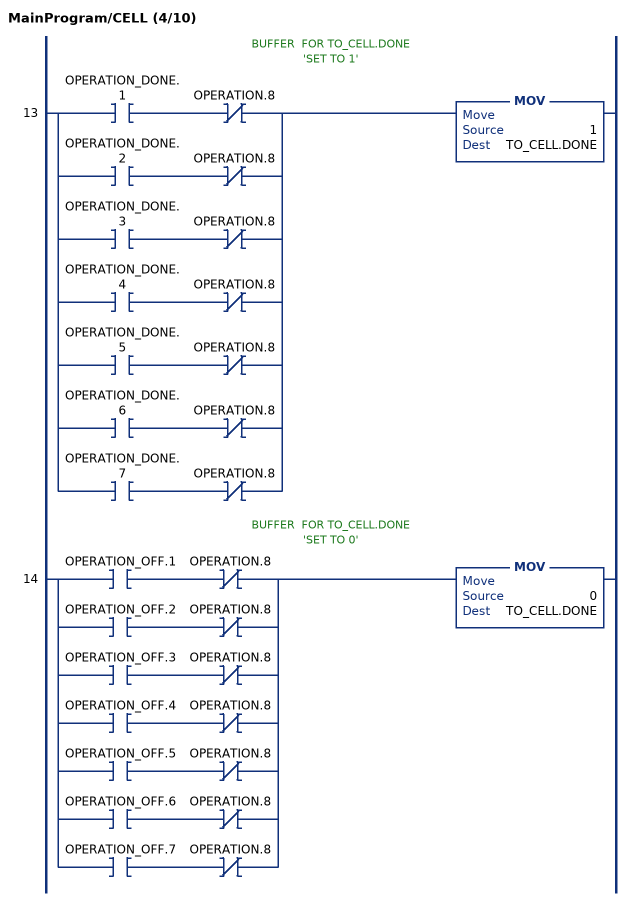
   // BUFFER  FOR TO_CELL.DONE
   // 'SET TO 1'
   13: [XIC(OPERATION_DONE.1) XIO(OPERATION.8) ,XIC(OPERATION_DONE.2) XIO(OPERATION.8) ,XIC(OPERATION_DONE.3) XIO(OPERATION.8) ,XIC(OPERATION_DONE.4) XIO(OPERATION.8) ,XIC(OPERATION_DONE.5) XIO(OPERATION.8) ,XIC(OPERATION_DONE.6) XIO(OPERATION.8) ,XIC(OPERATION_DONE.7) XIO(OPERATION.8) ]MOV(1,TO_CELL.DONE);
   // BUFFER  FOR TO_CELL.DONE
   // 'SET TO 0'
   14: [XIC(OPERATION_OFF.1) XIO(OPERATION.8) ,XIC(OPERATION_OFF.2) XIO(OPERATION.8) ,XIC(OPERATION_OFF.3) XIO(OPERATION.8) ,XIC(OPERATION_OFF.4) XIO(OPERATION.8) ,XIC(OPERATION_OFF.5) XIO(OPERATION.8) ,XIC(OPERATION_OFF.6) XIO(OPERATION.8) ,XIC(OPERATION_OFF.7) XIO(OPERATION.8) ]MOV(0,TO_CELL.DONE);
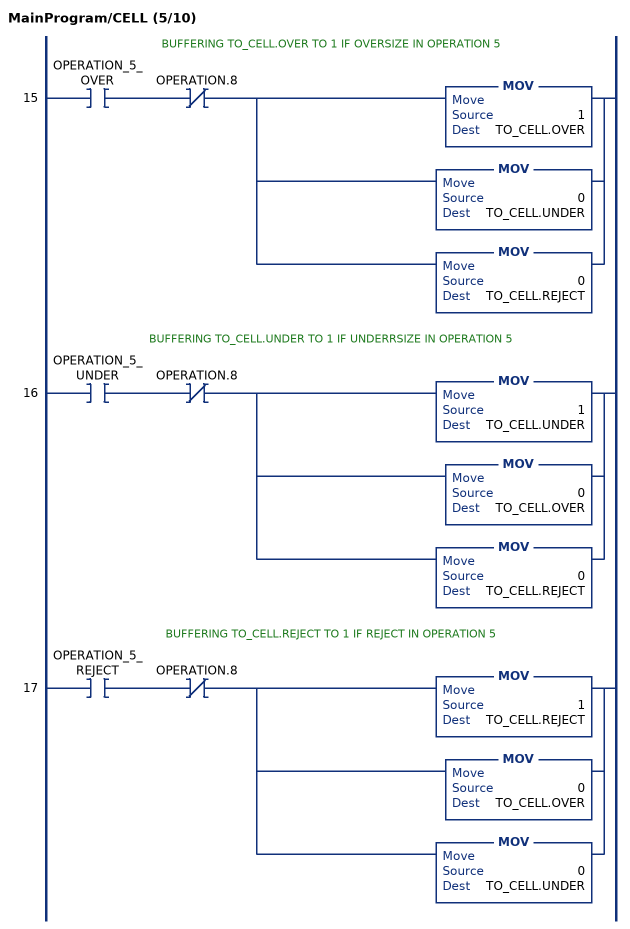
   // BUFFERING TO_CELL.OVER TO 1 IF OVERSIZE IN OPERATION 5
   15: XIC(OPERATION_5_OVER)XIO(OPERATION.8)[MOV(1,TO_CELL.OVER) ,MOV(0,TO_CELL.UNDER) ,MOV(0,TO_CELL.REJECT) ];
   // BUFFERING TO_CELL.UNDER TO 1 IF UNDERRSIZE IN OPERATION 5
   16: XIC(OPERATION_5_UNDER)XIO(OPERATION.8)[MOV(1,TO_CELL.UNDER) ,MOV(0,TO_CELL.OVER) ,MOV(0,TO_CELL.REJECT) ];
   // BUFFERING TO_CELL.REJECT TO 1 IF REJECT IN OPERATION 5
   17: XIC(OPERATION_5_REJECT)XIO(OPERATION.8)[MOV(1,TO_CELL.REJECT) ,MOV(0,TO_CELL.OVER) ,MOV(0,TO_CELL.UNDER) ];
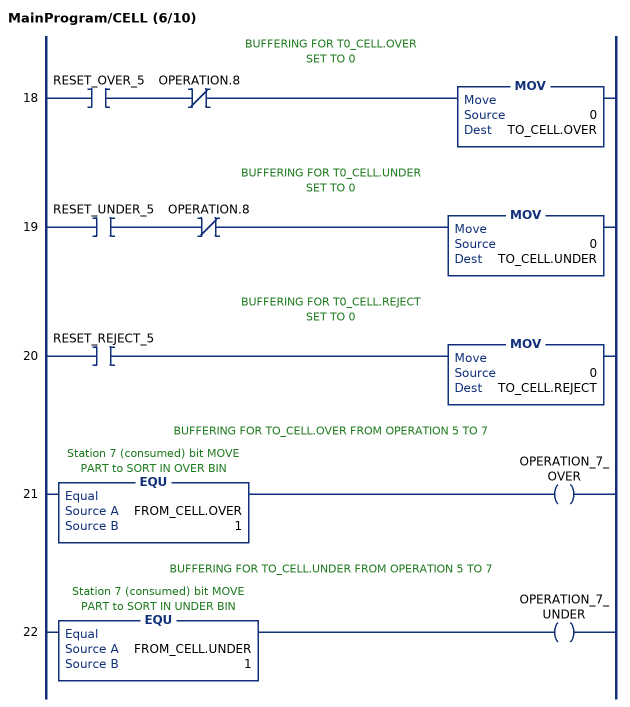
   // BUFFERING FOR T0_CELL.OVER
   // SET TO 0
   18: XIC(RESET_OVER_5)XIO(OPERATION.8)MOV(0,TO_CELL.OVER);
   // BUFFERING FOR T0_CELL.UNDER
   // SET TO 0
   19: XIC(RESET_UNDER_5)XIO(OPERATION.8)MOV(0,TO_CELL.UNDER);
   // BUFFERING FOR T0_CELL.REJECT
   // SET TO 0
   20: XIC(RESET_REJECT_5)MOV(0,TO_CELL.REJECT);
   // BUFFERING FOR TO_CELL.OVER FROM OPERATION 5 TO 7
   21: EQU(FROM_CELL.OVER,1)OTE(OPERATION_7_OVER);
   // BUFFERING FOR TO_CELL.UNDER FROM OPERATION 5 TO 7
   22: EQU(FROM_CELL.UNDER,1)OTE(OPERATION_7_UNDER);
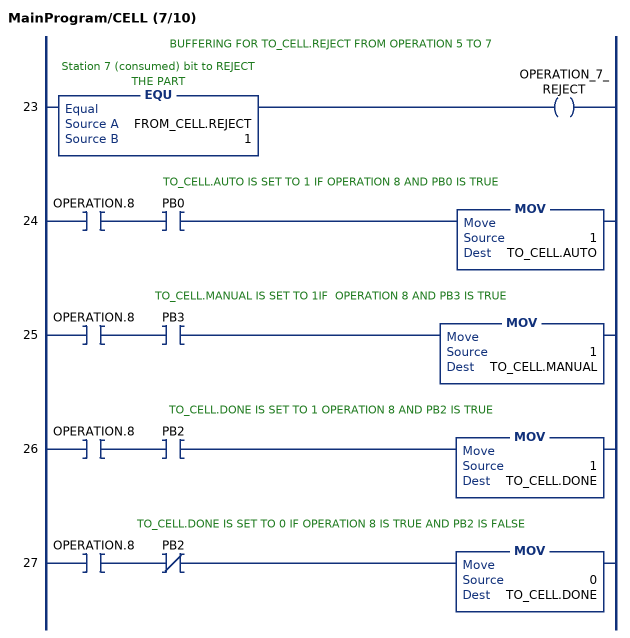
   // BUFFERING FOR TO_CELL.REJECT FROM OPERATION 5 TO 7
   23: EQU(FROM_CELL.REJECT,1)OTE(OPERATION_7_REJECT);
   // TO_CELL.AUTO IS SET TO 1 IF OPERATION 8 AND PB0 IS TRUE
   24: XIC(OPERATION.8)XIC(PB0)MOV(1,TO_CELL.AUTO);
   // TO_CELL.MANUAL IS SET TO 1IF  OPERATION 8 AND PB3 IS TRUE
   25: XIC(OPERATION.8)XIC(PB3)MOV(1,TO_CELL.MANUAL);
   // TO_CELL.DONE IS SET TO 1 OPERATION 8 AND PB2 IS TRUE
   26: XIC(OPERATION.8)XIC(PB2)MOV(1,TO_CELL.DONE);
   // TO_CELL.DONE IS SET TO 0 IF OPERATION 8 IS TRUE AND PB2 IS FALSE
   27: XIC(OPERATION.8)XIO(PB2)MOV(0,TO_CELL.DONE);
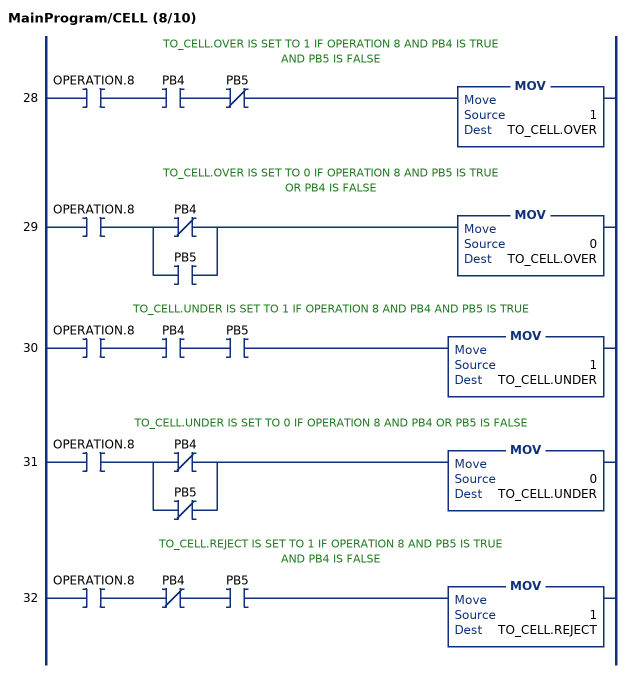
   // TO_CELL.OVER IS SET TO 1 IF OPERATION 8 AND PB4 IS TRUE
   // AND PB5 IS FALSE
   28: XIC(OPERATION.8)XIC(PB4)XIO(PB5)MOV(1,TO_CELL.OVER);
   // TO_CELL.OVER IS SET TO 0 IF OPERATION 8 AND PB5 IS TRUE
   // OR PB4 IS FALSE
   29: XIC(OPERATION.8)[XIO(PB4) ,XIC(PB5) ]MOV(0,TO_CELL.OVER);
   // TO_CELL.UNDER IS SET TO 1 IF OPERATION 8 AND PB4 AND PB5 IS TRUE
   30: XIC(OPERATION.8)XIC(PB4)XIC(PB5)MOV(1,TO_CELL.UNDER);
   // TO_CELL.UNDER IS SET TO 0 IF OPERATION 8 AND PB4 OR PB5 IS FALSE
   31: XIC(OPERATION.8)[XIO(PB4) ,XIO(PB5) ]MOV(0,TO_CELL.UNDER);
   // TO_CELL.REJECT IS SET TO 1 IF OPERATION 8 AND PB5 IS TRUE
   // AND PB4 IS FALSE
   32: XIC(OPERATION.8)XIO(PB4)XIC(PB5)MOV(1,TO_CELL.REJECT);
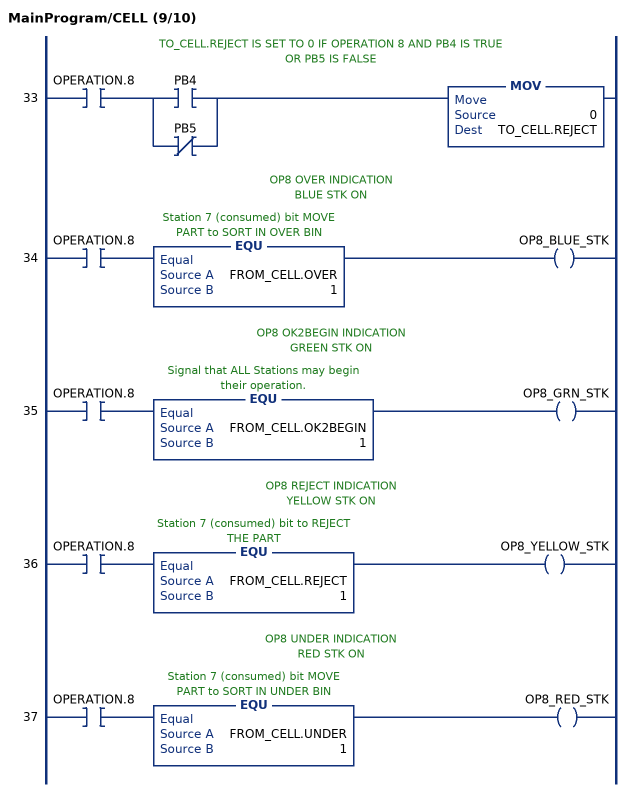
   // TO_CELL.REJECT IS SET TO 0 IF OPERATION 8 AND PB4 IS TRUE
   // OR PB5 IS FALSE
   33: XIC(OPERATION.8)[XIC(PB4) ,XIO(PB5) ]MOV(0,TO_CELL.REJECT);
   // OP8 OVER INDICATION
   // BLUE STK ON
   34: XIC(OPERATION.8)EQU(FROM_CELL.OVER,1)OTE(OP8_BLUE_STK);
   // OP8 OK2BEGIN INDICATION
   // GREEN STK ON
   35: XIC(OPERATION.8)EQU(FROM_CELL.OK2BEGIN,1)OTE(OP8_GRN_STK);
   // OP8 REJECT INDICATION
   // YELLOW STK ON
   36: XIC(OPERATION.8)EQU(FROM_CELL.REJECT,1)OTE(OP8_YELLOW_STK);
   // OP8 UNDER INDICATION
   // RED STK ON
   37: XIC(OPERATION.8)EQU(FROM_CELL.UNDER,1)OTE(OP8_RED_STK);
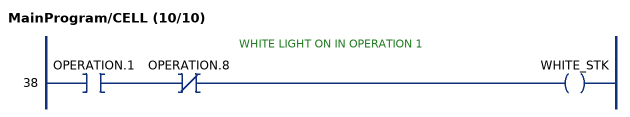
   // WHITE LIGHT ON IN OPERATION 1
   38: XIC(OPERATION.1)XIO(OPERATION.8)OTE(WHITE_STK);
END_ROUTINE

ROUTINE EXECUTION   (* ladder *)
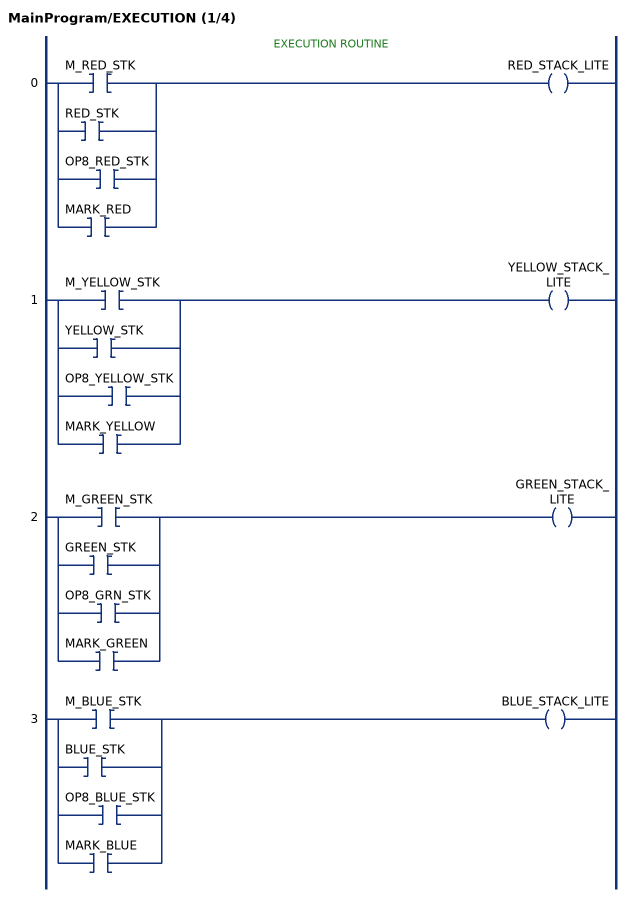
   // EXECUTION ROUTINE
   0: [XIC(M_RED_STK) ,XIC(RED_STK) ,XIC(OP8_RED_STK) ,XIC(MARK_RED) ]OTE(RED_STACK_LITE);
   1: [XIC(M_YELLOW_STK) ,XIC(YELLOW_STK) ,XIC(OP8_YELLOW_STK) ,XIC(MARK_YELLOW) ]OTE(YELLOW_STACK_LITE);
   2: [XIC(M_GREEN_STK) ,XIC(GREEN_STK) ,XIC(OP8_GRN_STK) ,XIC(MARK_GREEN) ]OTE(GREEN_STACK_LITE);
   3: [XIC(M_BLUE_STK) ,XIC(BLUE_STK) ,XIC(OP8_BLUE_STK) ,XIC(MARK_BLUE) ]OTE(BLUE_STACK_LITE);
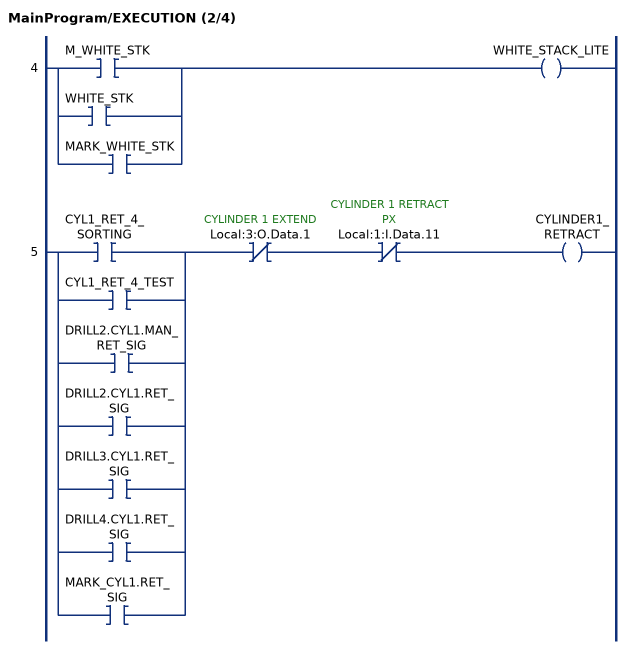
   4: [XIC(M_WHITE_STK) ,XIC(WHITE_STK) ,XIC(MARK_WHITE_STK) ]OTE(WHITE_STACK_LITE);
   5: [XIC(CYL1_RET_4_SORTING) ,XIC(CYL1_RET_4_TEST) ,XIC(DRILL2.CYL1.MAN_RET_SIG) ,XIC(DRILL2.CYL1.RET_SIG) ,XIC(DRILL3.CYL1.RET_SIG) ,XIC(DRILL4.CYL1.RET_SIG) ,XIC(MARK_CYL1.RET_SIG) ]XIO(Local:3:O.Data.1)XIO(Local:1:I.Data.11)OTE(CYLINDER1_RETRACT);
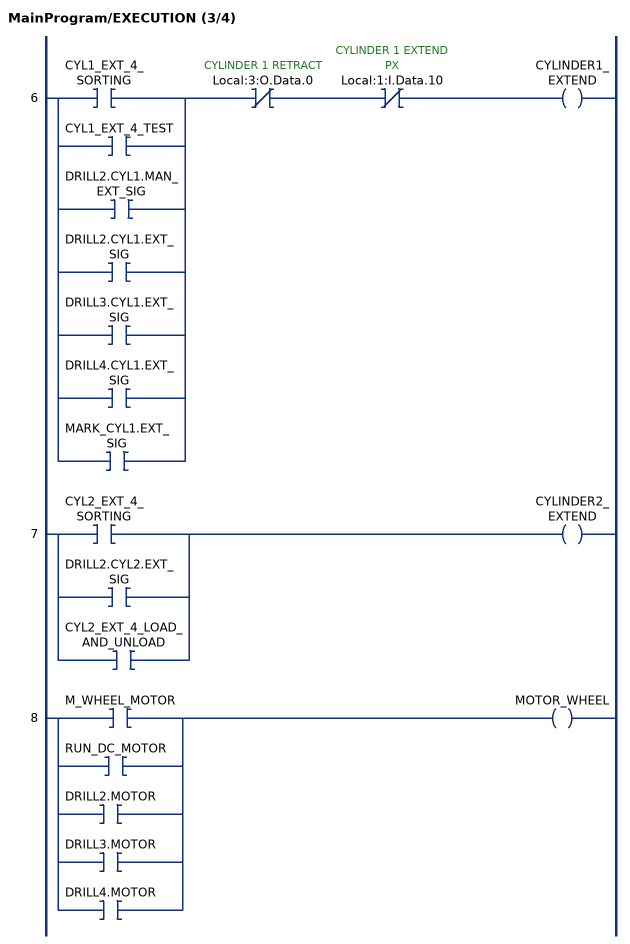
   6: [XIC(CYL1_EXT_4_SORTING) ,XIC(CYL1_EXT_4_TEST) ,XIC(DRILL2.CYL1.MAN_EXT_SIG) ,XIC(DRILL2.CYL1.EXT_SIG) ,XIC(DRILL3.CYL1.EXT_SIG) ,XIC(DRILL4.CYL1.EXT_SIG) ,XIC(MARK_CYL1.EXT_SIG) ]XIO(Local:3:O.Data.0)XIO(Local:1:I.Data.10)OTE(CYLINDER1_EXTEND);
   7: [XIC(CYL2_EXT_4_SORTING) ,XIC(DRILL2.CYL2.EXT_SIG) ,XIC(CYL2_EXT_4_LOAD_AND_UNLOAD) ]OTE(CYLINDER2_EXTEND);
   8: [XIC(M_WHEEL_MOTOR) ,XIC(RUN_DC_MOTOR) ,XIC(DRILL2.MOTOR) ,XIC(DRILL3.MOTOR) ,XIC(DRILL4.MOTOR) ]OTE(MOTOR_WHEEL);
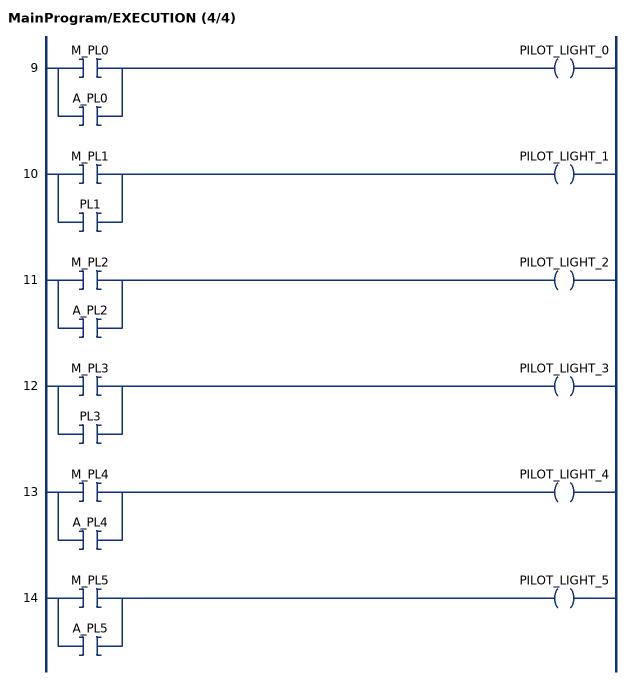
   9: [XIC(M_PL0) ,XIC(A_PL0) ]OTE(PILOT_LIGHT_0);
   10: [XIC(M_PL1) ,XIC(PL1) ]OTE(PILOT_LIGHT_1);
   11: [XIC(M_PL2) ,XIC(A_PL2) ]OTE(PILOT_LIGHT_2);
   12: [XIC(M_PL3) ,XIC(PL3) ]OTE(PILOT_LIGHT_3);
   13: [XIC(M_PL4) ,XIC(A_PL4) ]OTE(PILOT_LIGHT_4);
   14: [XIC(M_PL5) ,XIC(A_PL5) ]OTE(PILOT_LIGHT_5);
END_ROUTINE

ROUTINE FAULTS   (* ladder *)
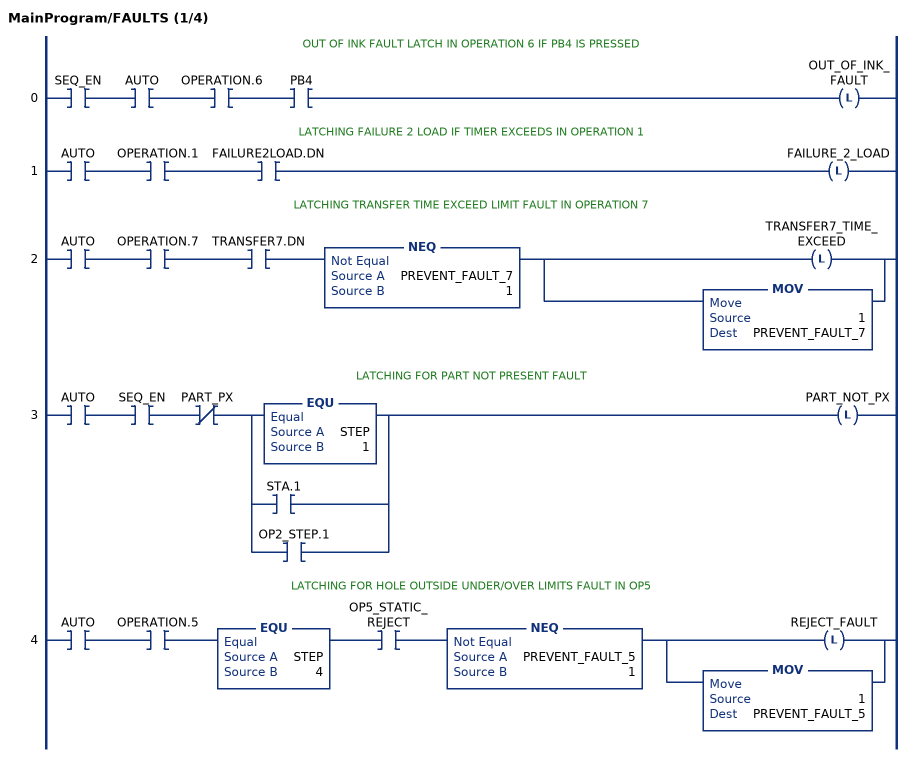
   // OUT OF INK FAULT LATCH IN OPERATION 6 IF PB4 IS PRESSED
   0: XIC(SEQ_EN)XIC(AUTO)XIC(OPERATION.6)XIC(PB4)OTL(OUT_OF_INK_FAULT);
   // LATCHING FAILURE 2 LOAD IF TIMER EXCEEDS IN OPERATION 1
   1: XIC(AUTO)XIC(OPERATION.1)XIC(FAILURE2LOAD.DN)OTL(FAILURE_2_LOAD);
   // LATCHING TRANSFER TIME EXCEED LIMIT FAULT IN OPERATION 7
   2: XIC(AUTO)XIC(OPERATION.7)XIC(TRANSFER7.DN)NEQ(PREVENT_FAULT_7,1)[OTL(TRANSFER7_TIME_EXCEED) ,MOV(1,PREVENT_FAULT_7) ];
   // LATCHING FOR PART NOT PRESENT FAULT
   3: XIC(AUTO)XIC(SEQ_EN)XIO(PART_PX)[EQU(STEP,1) ,XIC(STA.1) ,XIC(OP2_STEP.1) ]OTL(PART_NOT_PX);
   // LATCHING FOR HOLE OUTSIDE UNDER/OVER LIMITS FAULT IN OP5
   4: XIC(AUTO)XIC(OPERATION.5)EQU(STEP,4)XIC(OP5_STATIC_REJECT)NEQ(PREVENT_FAULT_5,1)[OTL(REJECT_FAULT) ,MOV(1,PREVENT_FAULT_5) ];
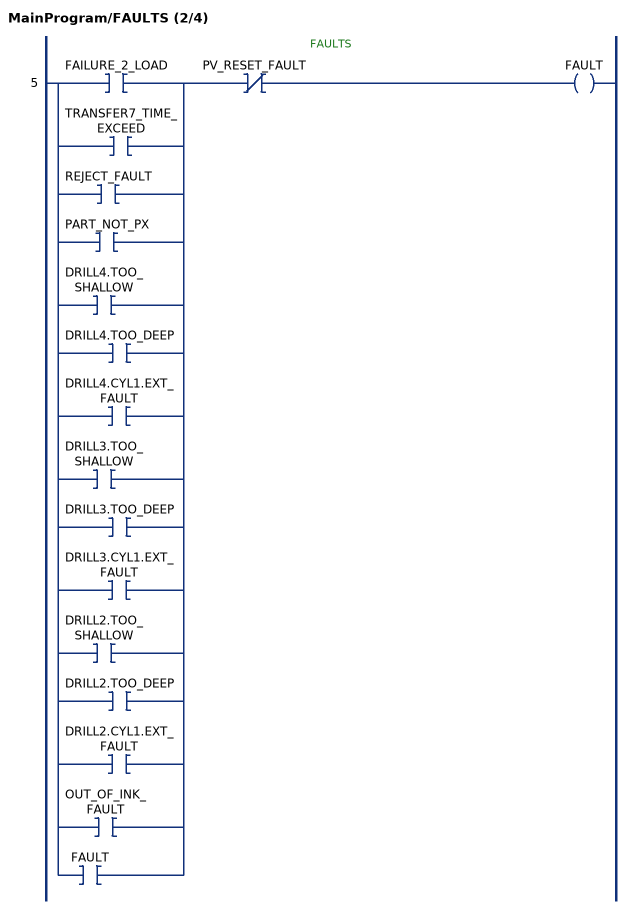
   // FAULTS
   5: [XIC(FAILURE_2_LOAD) ,XIC(TRANSFER7_TIME_EXCEED) ,XIC(REJECT_FAULT) ,XIC(PART_NOT_PX) ,XIC(DRILL4.TOO_SHALLOW) ,XIC(DRILL4.TOO_DEEP) ,XIC(DRILL4.CYL1.EXT_FAULT) ,XIC(DRILL3.TOO_SHALLOW) ,XIC(DRILL3.TOO_DEEP) ,XIC(DRILL3.CYL1.EXT_FAULT) ,XIC(DRILL2.TOO_SHALLOW) ,XIC(DRILL2.TOO_DEEP) ,XIC(DRILL2.CYL1.EXT_FAULT) ,XIC(OUT_OF_INK_FAULT) ,XIC(FAULT) ]XIO(PV_RESET_FAULT)OTE(FAULT);
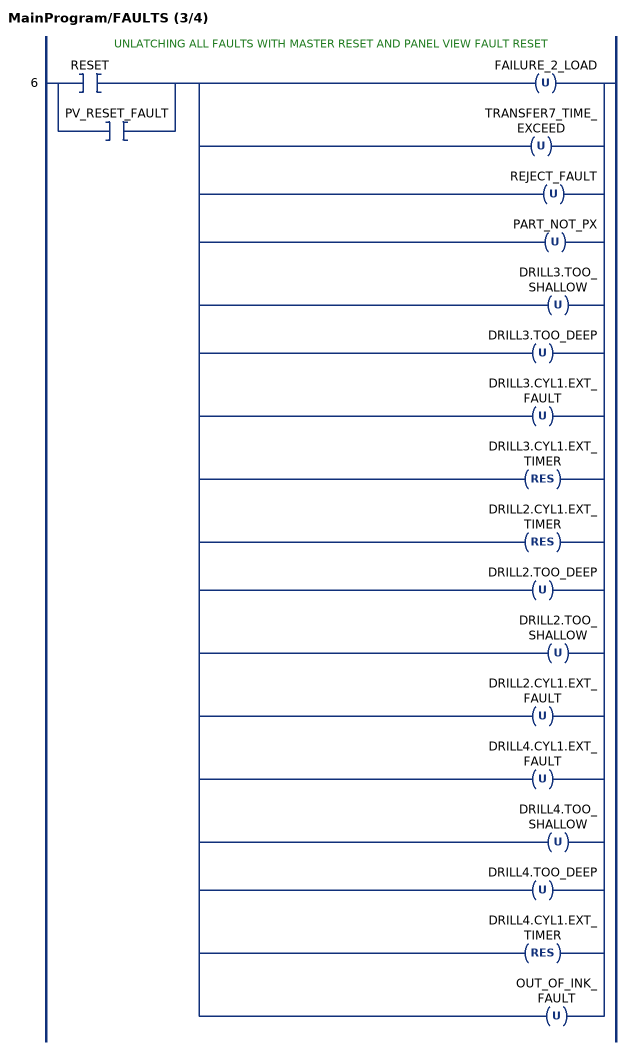
   // UNLATCHING ALL FAULTS WITH MASTER RESET AND PANEL VIEW FAULT RESET
   6: [XIC(RESET) ,XIC(PV_RESET_FAULT) ][OTU(FAILURE_2_LOAD) ,OTU(TRANSFER7_TIME_EXCEED) ,OTU(REJECT_FAULT) ,OTU(PART_NOT_PX) ,OTU(DRILL3.TOO_SHALLOW) ,OTU(DRILL3.TOO_DEEP) ,OTU(DRILL3.CYL1.EXT_FAULT) ,RES(DRILL3.CYL1.EXT_TIMER) ,RES(DRILL2.CYL1.EXT_TIMER) ,OTU(DRILL2.TOO_DEEP) ,OTU(DRILL2.TOO_SHALLOW) ,OTU(DRILL2.CYL1.EXT_FAULT) ,OTU(DRILL4.CYL1.EXT_FAULT) ,OTU(DRILL4.TOO_SHALLOW) ,OTU(DRILL4.TOO_DEEP) ,RES(DRILL4.CYL1.EXT_TIMER) ,OTU(OUT_OF_INK_FAULT) ];
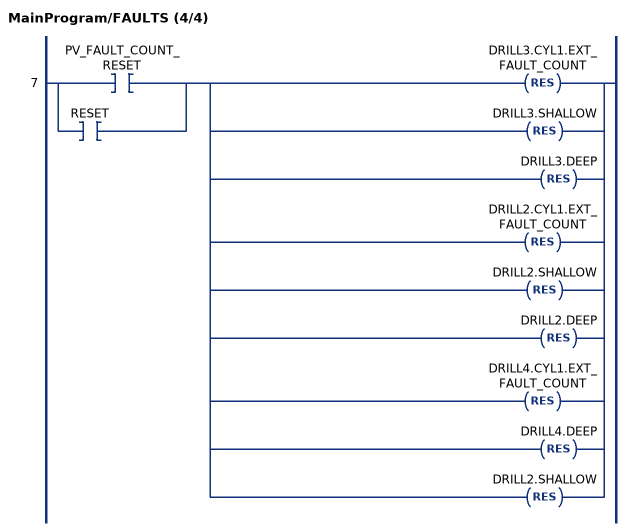
   7: [XIC(PV_FAULT_COUNT_RESET) ,XIC(RESET) ][RES(DRILL3.CYL1.EXT_FAULT_COUNT) ,RES(DRILL3.SHALLOW) ,RES(DRILL3.DEEP) ,RES(DRILL2.CYL1.EXT_FAULT_COUNT) ,RES(DRILL2.SHALLOW) ,RES(DRILL2.DEEP) ,RES(DRILL4.CYL1.EXT_FAULT_COUNT) ,RES(DRILL4.DEEP) ,RES(DRILL2.SHALLOW) ];
END_ROUTINE
